// TwinCAT 3 PLC project project
// ProgramVersion: 3.1.4023.0
// libraries:
//   Tc2_Standard, * (Beckhoff Automation GmbH)
//   Tc2_System, * (Beckhoff Automation GmbH)
//   Tc3_Module, * (Beckhoff Automation GmbH)
//   VisuSymbols,3.5.10.0,System
// project tree:
//   / GlobalTextList.TcGTLO, PlcTask.TcTTO, Visualization Manager.TcVMO (not stored)
//   POUs/ MAIN.TcPOU, POU.TcPOU
//   VISUs/ Visualization.TcVIS
// real-time tasks:
//   TASK PlcTask: cycle T#10ms, priority 20, ADS port 350

CONFIGURATION project
    RESOURCE PLC ON TwinCAT3
        TASK PlcTask(INTERVAL := T#10ms, PRIORITY := 20);
        PROGRAM MAIN WITH PlcTask : MAIN;
    END_RESOURCE
END_CONFIGURATION

// ---- POUs/MAIN.TcPOU
PROGRAM MAIN
VAR
END_VAR

POU();

END_PROGRAM

// ---- POUs/POU.TcPOU
PROGRAM POU
VAR
	
	A : BOOL := FALSE;
	B : BOOL := FALSE;
	C : BOOL := FALSE;
	D : BOOL := FALSE;

	TON_0: TON;
END_VAR

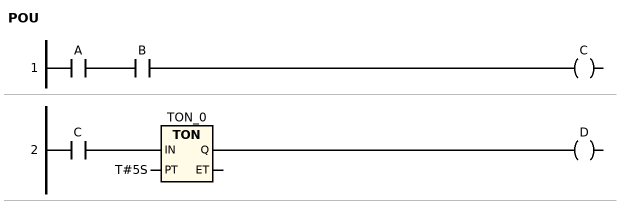
// NETWORK 1
C := A AND B;

// NETWORK 2
TON_0(IN := C, PT := T#5S); // TON
D := TON_0.Q;

END_PROGRAM

// ---- GlobalTextList.TcGTLO
TEXTLIST GlobalTextList
  550 = '%2.2f ms'
  332 = '%2.5f ms'
  127 = '%2.5f s'
  207 = 'A'
  487 = 'B'
  760 = 'C'
  768 = 'D'
  385 = 'Elapsed Time'
END_TEXTLIST

// ---- VISUs/Visualization.TcVIS
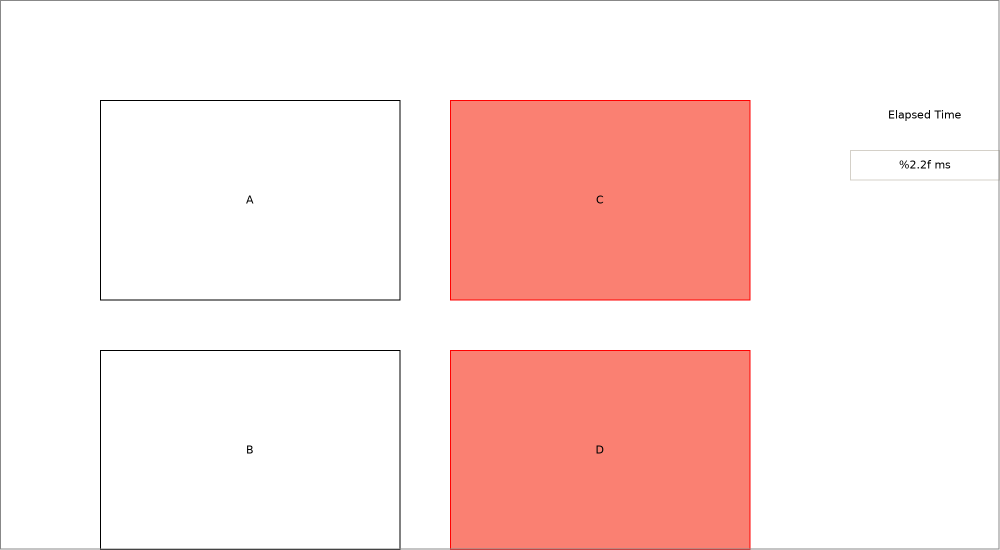
VISUALIZATION Visualization  // 1000x550
    RoundedRectangle (100,100 300x200), "A"
        OnMouseDown: toggle POU.A
    RoundedRectangle (100,350 300x200), "B"
        OnMouseDown: toggle POU.B
    RoundedRectangle (450,100 300x200), "C", colour toggle: POU.C
    RoundedRectangle (450,350 300x200), "D", colour toggle: POU.D
    Textfield (850,150 150x30), "%2.2f ms", text variable: POU.TON_0.ET
    Label (850,100 150x30), "Elapsed Time"
END_VISUALIZATION
